// TIA Portal V18 export
VAR_GLOBAL   // PLC tag table "20_AE2-SA3"
   "iAE2-SA3p" AT %I12.2 : Bool;   // 8
   "iAE2-SA3" AT %I12.3 : Bool;   // 8
   "iAE2-SA3a" AT %I17.7 : Bool;
   "oAE2-SA3p" AT %Q9.5 : Bool;
   "oAE2-SA3" AT %Q9.6 : Bool;
END_VAR
